SUBAPPLICATION Uebung_020h (* DigitalInput_I1 auf DigitalOutput_Q1; E_PULSE; Impulsformend *)
  (* Standard: 61499-2; Description: Copyright (c) 2023 Meisterschulen am Ostbahnhof This program and the accompanying materials are made available under the terms of the Eclipse Public License 2.0 which is available at https://www.eclipse.org/legal/epl-2.0/ SPDX-License-Identifier: EPL-2.0 *)
  (* Version 1.0, 2023-10-23, Franz Höpfinger, Meisterschulen am Ostbahnhof *)
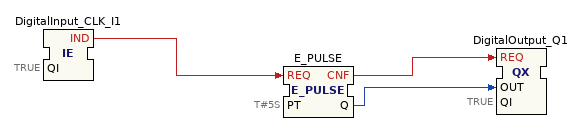
  FBS
    DigitalOutput_Q1 : QX(QI := TRUE);
    E_PULSE : E_PULSE(PT := T#5S);
    DigitalInput_CLK_I1 : IE(QI := TRUE);
  END_FBS
  EVENT_CONNECTIONS
    E_PULSE.CNF TO DigitalOutput_Q1.REQ;
    DigitalInput_CLK_I1.IND TO E_PULSE.REQ;
  END_CONNECTIONS
  DATA_CONNECTIONS
    E_PULSE.Q TO DigitalOutput_Q1.OUT;
  END_CONNECTIONS
END_SUBAPPLICATION
